// Returns True if the response indicates success.
FUNCTION _F_IsSuccessfulResponse : BOOL
VAR_INPUT
	jsonDoc : SJsonValue;
END_VAR
VAR
	fbJson : FB_JsonDomParser;
	jsonProp : SJsonValue;
END_VAR

IF NOT fbJson.HasMember(jsonDoc, 'status') THEN
	_F_IsSuccessfulResponse := FALSE;
	RETURN;
END_IF

jsonProp := fbJson.FindMember(jsonDoc, 'status');
_F_IsSuccessfulResponse := fbJson.GetBool(jsonProp);

END_FUNCTION

(* stored: Version 1.1.0.1
   POU _F_IsSuccessfulResponse: Id {29004567-fb11-4efd-bb26-c96ffa7dcf47}, SpecialFunc None *)
